// TIA Portal project "Proyecto_Dosificador_Mezclador_Automatico" (V17)

(* hardware
DEVICE "S7-1200 station_1"  S7-1200 Station
   slot 0: "Rack_0"  S7-1200 Rack  Rack  V1.0
   slot 1: "PLC_1"  CPU 1215C DC/DC/DC  6ES7 215-1AG40-0XB0  V4.5
*)

// ===== PLC "PLC_1"  CPU 1215C DC/DC/DC =====

VAR_GLOBAL   // PLC tag table "Default tag table"
   "System_Byte" AT %MB8190 : Byte;
   "FirstScan" AT %M8190.0 : Bool;
   "DiagStatusUpdate" AT %M8190.1 : Bool;
   "AlwaysTRUE" AT %M8190.2 : Bool;
   "AlwaysFALSE" AT %M8190.3 : Bool;
   "Clock_Byte" AT %MB8191 : Byte;
   "Clock_10Hz" AT %M8191.0 : Bool;
   "Clock_5Hz" AT %M8191.1 : Bool;
   "Clock_2.5Hz" AT %M8191.2 : Bool;
   "Clock_2Hz" AT %M8191.3 : Bool;
   "Clock_1.25Hz" AT %M8191.4 : Bool;
   "Clock_1Hz" AT %M8191.5 : Bool;
   "Clock_0.625Hz" AT %M8191.6 : Bool;
   "Clock_0.5Hz" AT %M8191.7 : Bool;
END_VAR

VAR_GLOBAL   // PLC tag table "Entradas"
   "Sel Funcionamiento" AT %I0.0 : Bool;
   "P Marcha NO" AT %I0.1 : Bool;
   "P Paro NC" AT %I0.2 : Bool;
   "P Emergencia NC" AT %I0.3 : Bool;
   "P Rearme NO" AT %I0.4 : Bool;
   "S Mezclador Nivel Bajo NC" AT %I0.5 : Bool;
   "S Briquetas NO" AT %I0.6 : Bool;
   "S FC Pivotante Arriba NC" AT %I0.7 : Bool;
   "S FC Pivotante Abajo NC" AT %I1.0 : Bool;
   "GM Cinta NC" AT %I1.1 : Bool;
   "GM Agitador NC" AT %I1.2 : Bool;
   "GM Pivotante NC" AT %I1.3 : Bool;
   "S Peso" AT %IW64 : Word;
END_VAR

VAR_GLOBAL   // PLC tag table "Salidas"
   "EV A Monoestable NC" AT %I1.6 : Bool;
   "EV B Monoestable NC" AT %I1.7 : Bool;
   "EV C Monoestable NC" AT %I2.0 : Bool;
   "M Cinta" AT %I2.1 : Bool;
   "M Agitador" AT %I2.2 : Bool;
   "M Pivotante Subir" AT %I2.3 : Bool;
   "M Pivotante Bajar" AT %I2.4 : Bool;
END_VAR

VAR_GLOBAL   // PLC tag table "Marcas Generales"
   "S Peso Normalizado" AT %MD2000 : Real;
   "S Peso Escalado" AT %MD2004 : Real;
   "Marca Marcha NO" AT %M2008.0 : Bool;
   "Marca Paro NC" AT %M2008.1 : Bool;
   "Marca Seguridad NC" AT %M2008.2 : Bool;
   "Marca Rearme NO" AT %M2008.3 : Bool;
   "Marca Sel Funcionamiento" AT %M2008.4 : Bool;
   "Marca Sel Mantenimiento" AT %M2008.5 : Bool;
   "Marca CI Todas" AT %M2008.6 : Bool;
   "Marca Etapas Iniciales" AT %M2008.7 : Bool;
   "Marca CI Mezclador" AT %M2009.0 : Bool;
   "Marca CI Depositos" AT %M2009.1 : Bool;
   "Marca CI Briquetas" AT %M2009.2 : Bool;
   "Marca CI Electrovalvulas" AT %M2009.3 : Bool;
END_VAR

VAR_GLOBAL   // PLC tag table "Etapas"
   "E0" AT %M0.0 : Bool;   // Etapas funcionamiento E0-E99
   "E1" AT %M0.1 : Bool;   // Etapas funcionamiento E0-E99
   "E2" AT %M0.2 : Bool;   // Etapas funcionamiento E0-E99
   "E3" AT %M0.3 : Bool;   // Etapas funcionamiento E0-E99
   "E4" AT %M0.4 : Bool;   // Etapas funcionamiento E0-E99
   "E5" AT %M0.5 : Bool;   // Etapas funcionamiento E0-E99
   "E6" AT %M0.6 : Bool;   // Etapas funcionamiento E0-E99
   "E7" AT %M0.7 : Bool;   // Etapas funcionamiento E0-E99
   "E8" AT %M1.0 : Bool;   // Etapas funcionamiento E0-E99
   "E9" AT %M1.1 : Bool;   // Etapas funcionamiento E0-E99
   "E10" AT %M1.2 : Bool;   // Etapas funcionamiento E0-E99
   "E11" AT %M1.3 : Bool;   // Etapas funcionamiento E0-E99
   "E12" AT %M1.4 : Bool;   // Etapas funcionamiento E0-E99
   "E13" AT %M1.5 : Bool;   // Etapas funcionamiento E0-E99
   "E14" AT %M1.6 : Bool;   // Etapas funcionamiento E0-E99
   "E15" AT %M1.7 : Bool;   // Etapas funcionamiento E0-E99
   "E16" AT %M2.0 : Bool;   // Etapas funcionamiento E0-E99
   "E17" AT %M2.1 : Bool;   // Etapas funcionamiento E0-E99
   "E18" AT %M2.2 : Bool;   // Etapas funcionamiento E0-E99
   "E19" AT %M2.3 : Bool;   // Etapas funcionamiento E0-E99
   "E20" AT %M2.4 : Bool;   // Etapas funcionamiento E0-E99
   "E21" AT %M2.5 : Bool;   // Etapas funcionamiento E0-E99
   "E22" AT %M2.6 : Bool;   // Etapas funcionamiento E0-E99
   "E23" AT %M2.7 : Bool;   // Etapas funcionamiento E0-E99
   "E24" AT %M3.0 : Bool;   // Etapas funcionamiento E0-E99
   "E25" AT %M3.1 : Bool;   // Etapas funcionamiento E0-E99
   "E26" AT %M3.2 : Bool;   // Etapas funcionamiento E0-E99
   "E27" AT %M3.3 : Bool;   // Etapas funcionamiento E0-E99
   "E28" AT %M3.4 : Bool;   // Etapas funcionamiento E0-E99
   "E29" AT %M3.5 : Bool;   // Etapas funcionamiento E0-E99
   "E30" AT %M3.6 : Bool;   // Etapas funcionamiento E0-E99
   "E31" AT %M3.7 : Bool;   // Etapas funcionamiento E0-E99
   "E32" AT %M4.0 : Bool;   // Etapas funcionamiento E0-E99
   "E33" AT %M4.1 : Bool;   // Etapas funcionamiento E0-E99
   "E34" AT %M4.2 : Bool;   // Etapas funcionamiento E0-E99
   "E35" AT %M4.3 : Bool;   // Etapas funcionamiento E0-E99
   "E36" AT %M4.4 : Bool;   // Etapas funcionamiento E0-E99
   "E37" AT %M4.5 : Bool;   // Etapas funcionamiento E0-E99
   "E38" AT %M4.6 : Bool;   // Etapas funcionamiento E0-E99
   "E39" AT %M4.7 : Bool;   // Etapas funcionamiento E0-E99
   "E40" AT %M5.0 : Bool;   // Etapas funcionamiento E0-E99
   "E41" AT %M5.1 : Bool;   // Etapas funcionamiento E0-E99
   "E42" AT %M5.2 : Bool;   // Etapas funcionamiento E0-E99
   "E43" AT %M5.3 : Bool;   // Etapas funcionamiento E0-E99
   "E44" AT %M5.4 : Bool;   // Etapas funcionamiento E0-E99
   "E45" AT %M5.5 : Bool;   // Etapas funcionamiento E0-E99
   "E46" AT %M5.6 : Bool;   // Etapas funcionamiento E0-E99
   "E47" AT %M5.7 : Bool;   // Etapas funcionamiento E0-E99
   "E48" AT %M6.0 : Bool;   // Etapas funcionamiento E0-E99
   "E49" AT %M6.1 : Bool;   // Etapas funcionamiento E0-E99
   "E50" AT %M6.2 : Bool;   // Etapas funcionamiento E0-E99
   "E51" AT %M6.3 : Bool;   // Etapas funcionamiento E0-E99
   "E52" AT %M6.4 : Bool;   // Etapas funcionamiento E0-E99
   "E53" AT %M6.5 : Bool;   // Etapas funcionamiento E0-E99
   "E54" AT %M6.6 : Bool;   // Etapas funcionamiento E0-E99
   "E55" AT %M6.7 : Bool;   // Etapas funcionamiento E0-E99
   "E56" AT %M7.0 : Bool;   // Etapas funcionamiento E0-E99
   "E57" AT %M7.1 : Bool;   // Etapas funcionamiento E0-E99
   "E58" AT %M7.2 : Bool;   // Etapas funcionamiento E0-E99
   "E59" AT %M7.3 : Bool;   // Etapas funcionamiento E0-E99
   "E60" AT %M7.4 : Bool;   // Etapas funcionamiento E0-E99
   "E61" AT %M7.5 : Bool;   // Etapas funcionamiento E0-E99
   "E62" AT %M7.6 : Bool;   // Etapas funcionamiento E0-E99
   "E63" AT %M7.7 : Bool;   // Etapas funcionamiento E0-E99
   "E64" AT %M8.0 : Bool;   // Etapas funcionamiento E0-E99
   "E65" AT %M8.1 : Bool;   // Etapas funcionamiento E0-E99
   "E66" AT %M8.2 : Bool;   // Etapas funcionamiento E0-E99
   "E67" AT %M8.3 : Bool;   // Etapas funcionamiento E0-E99
   "E68" AT %M8.4 : Bool;   // Etapas funcionamiento E0-E99
   "E69" AT %M8.5 : Bool;   // Etapas funcionamiento E0-E99
   "E70" AT %M8.6 : Bool;   // Etapas funcionamiento E0-E99
   "E71" AT %M8.7 : Bool;   // Etapas funcionamiento E0-E99
   "E72" AT %M9.0 : Bool;   // Etapas funcionamiento E0-E99
   "E73" AT %M9.1 : Bool;   // Etapas funcionamiento E0-E99
   "E74" AT %M9.2 : Bool;   // Etapas funcionamiento E0-E99
   "E75" AT %M9.3 : Bool;   // Etapas funcionamiento E0-E99
   "E76" AT %M9.4 : Bool;   // Etapas funcionamiento E0-E99
   "E77" AT %M9.5 : Bool;   // Etapas funcionamiento E0-E99
   "E78" AT %M9.6 : Bool;   // Etapas funcionamiento E0-E99
   "E79" AT %M9.7 : Bool;   // Etapas funcionamiento E0-E99
   "E80" AT %M10.0 : Bool;   // Etapas funcionamiento E0-E99
   "E81" AT %M10.1 : Bool;   // Etapas funcionamiento E0-E99
   "E82" AT %M10.2 : Bool;   // Etapas funcionamiento E0-E99
   "E83" AT %M10.3 : Bool;   // Etapas funcionamiento E0-E99
   "E84" AT %M10.4 : Bool;   // Etapas funcionamiento E0-E99
   "E85" AT %M10.5 : Bool;   // Etapas funcionamiento E0-E99
   "E86" AT %M10.6 : Bool;   // Etapas funcionamiento E0-E99
   "E87" AT %M10.7 : Bool;   // Etapas funcionamiento E0-E99
   "E88" AT %M11.0 : Bool;   // Etapas funcionamiento E0-E99
   "E89" AT %M11.1 : Bool;   // Etapas funcionamiento E0-E99
   "E90" AT %M11.2 : Bool;   // Etapas funcionamiento E0-E99
   "E91" AT %M11.3 : Bool;   // Etapas funcionamiento E0-E99
   "E92" AT %M11.4 : Bool;   // Etapas funcionamiento E0-E99
   "E93" AT %M11.5 : Bool;   // Etapas funcionamiento E0-E99
   "E94" AT %M11.6 : Bool;   // Etapas funcionamiento E0-E99
   "E95" AT %M11.7 : Bool;   // Etapas funcionamiento E0-E99
   "E96" AT %M12.0 : Bool;   // Etapas funcionamiento E0-E99
   "E97" AT %M12.1 : Bool;   // Etapas funcionamiento E0-E99
   "E98" AT %M12.2 : Bool;   // Etapas funcionamiento E0-E99
   "E99" AT %M12.3 : Bool;   // Etapas funcionamiento E0-E99
   "E100" AT %M100.0 : Bool;   // Etapas modos marcha E100-E199
   "E101" AT %M100.1 : Bool;   // Etapas modos marcha E100-E199
   "E102" AT %M100.2 : Bool;   // Etapas modos marcha E100-E199
   "E103" AT %M100.3 : Bool;   // Etapas modos marcha E100-E199
   "E104" AT %M100.4 : Bool;   // Etapas modos marcha E100-E199
   "E105" AT %M100.5 : Bool;   // Etapas modos marcha E100-E199
   "E106" AT %M100.6 : Bool;   // Etapas modos marcha E100-E199
   "E107" AT %M100.7 : Bool;   // Etapas modos marcha E100-E199
   "E108" AT %M101.0 : Bool;   // Etapas modos marcha E100-E199
   "E109" AT %M101.1 : Bool;   // Etapas modos marcha E100-E199
   "E110" AT %M101.2 : Bool;   // Etapas modos marcha E100-E199
   "E111" AT %M101.3 : Bool;   // Etapas modos marcha E100-E199
   "E112" AT %M101.4 : Bool;   // Etapas modos marcha E100-E199
   "E113" AT %M101.5 : Bool;   // Etapas modos marcha E100-E199
   "E114" AT %M101.6 : Bool;   // Etapas modos marcha E100-E199
   "E115" AT %M101.7 : Bool;   // Etapas modos marcha E100-E199
   "E116" AT %M102.0 : Bool;   // Etapas modos marcha E100-E199
   "E117" AT %M102.1 : Bool;   // Etapas modos marcha E100-E199
   "E118" AT %M102.2 : Bool;   // Etapas modos marcha E100-E199
   "E119" AT %M102.3 : Bool;   // Etapas modos marcha E100-E199
   "E120" AT %M102.4 : Bool;   // Etapas modos marcha E100-E199
   "E121" AT %M102.5 : Bool;   // Etapas modos marcha E100-E199
   "E122" AT %M102.6 : Bool;   // Etapas modos marcha E100-E199
   "E123" AT %M102.7 : Bool;   // Etapas modos marcha E100-E199
   "E124" AT %M103.0 : Bool;   // Etapas modos marcha E100-E199
   "E125" AT %M103.1 : Bool;   // Etapas modos marcha E100-E199
   "E126" AT %M103.2 : Bool;   // Etapas modos marcha E100-E199
   "E127" AT %M103.3 : Bool;   // Etapas modos marcha E100-E199
   "E128" AT %M103.4 : Bool;   // Etapas modos marcha E100-E199
   "E129" AT %M103.5 : Bool;   // Etapas modos marcha E100-E199
   "E130" AT %M103.6 : Bool;   // Etapas modos marcha E100-E199
   "E131" AT %M103.7 : Bool;   // Etapas modos marcha E100-E199
   "E132" AT %M104.0 : Bool;   // Etapas modos marcha E100-E199
   "E133" AT %M104.1 : Bool;   // Etapas modos marcha E100-E199
   "E134" AT %M104.2 : Bool;   // Etapas modos marcha E100-E199
   "E135" AT %M104.3 : Bool;   // Etapas modos marcha E100-E199
   "E136" AT %M104.4 : Bool;   // Etapas modos marcha E100-E199
   "E137" AT %M104.5 : Bool;   // Etapas modos marcha E100-E199
   "E138" AT %M104.6 : Bool;   // Etapas modos marcha E100-E199
   "E139" AT %M104.7 : Bool;   // Etapas modos marcha E100-E199
   "E140" AT %M105.0 : Bool;   // Etapas modos marcha E100-E199
   "E141" AT %M105.1 : Bool;   // Etapas modos marcha E100-E199
   "E142" AT %M105.2 : Bool;   // Etapas modos marcha E100-E199
   "E143" AT %M105.3 : Bool;   // Etapas modos marcha E100-E199
   "E144" AT %M105.4 : Bool;   // Etapas modos marcha E100-E199
   "E145" AT %M105.5 : Bool;   // Etapas modos marcha E100-E199
   "E146" AT %M105.6 : Bool;   // Etapas modos marcha E100-E199
   "E147" AT %M105.7 : Bool;   // Etapas modos marcha E100-E199
   "E148" AT %M106.0 : Bool;   // Etapas modos marcha E100-E199
   "E149" AT %M106.1 : Bool;   // Etapas modos marcha E100-E199
   "E150" AT %M106.2 : Bool;   // Etapas modos marcha E100-E199
   "E151" AT %M106.3 : Bool;   // Etapas modos marcha E100-E199
   "E152" AT %M106.4 : Bool;   // Etapas modos marcha E100-E199
   "E153" AT %M106.5 : Bool;   // Etapas modos marcha E100-E199
   "E154" AT %M106.6 : Bool;   // Etapas modos marcha E100-E199
   "E155" AT %M106.7 : Bool;   // Etapas modos marcha E100-E199
   "E156" AT %M107.0 : Bool;   // Etapas modos marcha E100-E199
   "E157" AT %M107.1 : Bool;   // Etapas modos marcha E100-E199
   "E158" AT %M107.2 : Bool;   // Etapas modos marcha E100-E199
   "E159" AT %M107.3 : Bool;   // Etapas modos marcha E100-E199
   "E160" AT %M107.4 : Bool;   // Etapas modos marcha E100-E199
   "E161" AT %M107.5 : Bool;   // Etapas modos marcha E100-E199
   "E162" AT %M107.6 : Bool;   // Etapas modos marcha E100-E199
   "E163" AT %M107.7 : Bool;   // Etapas modos marcha E100-E199
   "E164" AT %M108.0 : Bool;   // Etapas modos marcha E100-E199
   "E165" AT %M108.1 : Bool;   // Etapas modos marcha E100-E199
   "E166" AT %M108.2 : Bool;   // Etapas modos marcha E100-E199
   "E167" AT %M108.3 : Bool;   // Etapas modos marcha E100-E199
   "E168" AT %M108.4 : Bool;   // Etapas modos marcha E100-E199
   "E169" AT %M108.5 : Bool;   // Etapas modos marcha E100-E199
   "E170" AT %M108.6 : Bool;   // Etapas modos marcha E100-E199
   "E171" AT %M108.7 : Bool;   // Etapas modos marcha E100-E199
   "E172" AT %M109.0 : Bool;   // Etapas modos marcha E100-E199
   "E173" AT %M109.1 : Bool;   // Etapas modos marcha E100-E199
   "E174" AT %M109.2 : Bool;   // Etapas modos marcha E100-E199
   "E175" AT %M109.3 : Bool;   // Etapas modos marcha E100-E199
   "E176" AT %M109.4 : Bool;   // Etapas modos marcha E100-E199
   "E177" AT %M109.5 : Bool;   // Etapas modos marcha E100-E199
   "E178" AT %M109.6 : Bool;   // Etapas modos marcha E100-E199
   "E179" AT %M109.7 : Bool;   // Etapas modos marcha E100-E199
   "E180" AT %M110.0 : Bool;   // Etapas modos marcha E100-E199
   "E181" AT %M110.1 : Bool;   // Etapas modos marcha E100-E199
   "E182" AT %M110.2 : Bool;   // Etapas modos marcha E100-E199
   "E183" AT %M110.3 : Bool;   // Etapas modos marcha E100-E199
   "E184" AT %M110.4 : Bool;   // Etapas modos marcha E100-E199
   "E185" AT %M110.5 : Bool;   // Etapas modos marcha E100-E199
   "E186" AT %M110.6 : Bool;   // Etapas modos marcha E100-E199
   "E187" AT %M110.7 : Bool;   // Etapas modos marcha E100-E199
   "E188" AT %M111.0 : Bool;   // Etapas modos marcha E100-E199
   "E189" AT %M111.1 : Bool;   // Etapas modos marcha E100-E199
   "E190" AT %M111.2 : Bool;   // Etapas modos marcha E100-E199
   "E191" AT %M111.3 : Bool;   // Etapas modos marcha E100-E199
   "E192" AT %M111.4 : Bool;   // Etapas modos marcha E100-E199
   "E193" AT %M111.5 : Bool;   // Etapas modos marcha E100-E199
   "E194" AT %M111.6 : Bool;   // Etapas modos marcha E100-E199
   "E195" AT %M111.7 : Bool;   // Etapas modos marcha E100-E199
   "E196" AT %M112.0 : Bool;   // Etapas modos marcha E100-E199
   "E197" AT %M112.1 : Bool;   // Etapas modos marcha E100-E199
   "E198" AT %M112.2 : Bool;   // Etapas modos marcha E100-E199
   "E199" AT %M112.3 : Bool;   // Etapas modos marcha E100-E199
   "E200" AT %M200.0 : Bool;   // Etapas condiciones iniciales E200-E299
   "E201" AT %M200.1 : Bool;   // Etapas condiciones iniciales E200-E299
   "E202" AT %M200.2 : Bool;   // Etapas condiciones iniciales E200-E299
   "E203" AT %M200.3 : Bool;   // Etapas condiciones iniciales E200-E299
   "E204" AT %M200.4 : Bool;   // Etapas condiciones iniciales E200-E299
   "E205" AT %M200.5 : Bool;   // Etapas condiciones iniciales E200-E299
   "E206" AT %M200.6 : Bool;   // Etapas condiciones iniciales E200-E299
   "E207" AT %M200.7 : Bool;   // Etapas condiciones iniciales E200-E299
   "E208" AT %M201.0 : Bool;   // Etapas condiciones iniciales E200-E299
   "E209" AT %M201.1 : Bool;   // Etapas condiciones iniciales E200-E299
   "E210" AT %M201.2 : Bool;   // Etapas condiciones iniciales E200-E299
   "E211" AT %M201.3 : Bool;   // Etapas condiciones iniciales E200-E299
   "E212" AT %M201.4 : Bool;   // Etapas condiciones iniciales E200-E299
   "E213" AT %M201.5 : Bool;   // Etapas condiciones iniciales E200-E299
   "E214" AT %M201.6 : Bool;   // Etapas condiciones iniciales E200-E299
   "E215" AT %M201.7 : Bool;   // Etapas condiciones iniciales E200-E299
   "E216" AT %M202.0 : Bool;   // Etapas condiciones iniciales E200-E299
   "E217" AT %M202.1 : Bool;   // Etapas condiciones iniciales E200-E299
   "E218" AT %M202.2 : Bool;   // Etapas condiciones iniciales E200-E299
   "E219" AT %M202.3 : Bool;   // Etapas condiciones iniciales E200-E299
   "E220" AT %M202.4 : Bool;   // Etapas condiciones iniciales E200-E299
   "E221" AT %M202.5 : Bool;   // Etapas condiciones iniciales E200-E299
   "E222" AT %M202.6 : Bool;   // Etapas condiciones iniciales E200-E299
   "E223" AT %M202.7 : Bool;   // Etapas condiciones iniciales E200-E299
   "E224" AT %M203.0 : Bool;   // Etapas condiciones iniciales E200-E299
   "E225" AT %M203.1 : Bool;   // Etapas condiciones iniciales E200-E299
   "E226" AT %M203.2 : Bool;   // Etapas condiciones iniciales E200-E299
   "E227" AT %M203.3 : Bool;   // Etapas condiciones iniciales E200-E299
   "E228" AT %M203.4 : Bool;   // Etapas condiciones iniciales E200-E299
   "E229" AT %M203.5 : Bool;   // Etapas condiciones iniciales E200-E299
   "E230" AT %M203.6 : Bool;   // Etapas condiciones iniciales E200-E299
   "E231" AT %M203.7 : Bool;   // Etapas condiciones iniciales E200-E299
   "E232" AT %M204.0 : Bool;   // Etapas condiciones iniciales E200-E299
   "E233" AT %M204.1 : Bool;   // Etapas condiciones iniciales E200-E299
   "E234" AT %M204.2 : Bool;   // Etapas condiciones iniciales E200-E299
   "E235" AT %M204.3 : Bool;   // Etapas condiciones iniciales E200-E299
   "E236" AT %M204.4 : Bool;   // Etapas condiciones iniciales E200-E299
   "E237" AT %M204.5 : Bool;   // Etapas condiciones iniciales E200-E299
   "E238" AT %M204.6 : Bool;   // Etapas condiciones iniciales E200-E299
   "E239" AT %M204.7 : Bool;   // Etapas condiciones iniciales E200-E299
   "E240" AT %M205.0 : Bool;   // Etapas condiciones iniciales E200-E299
   "E241" AT %M205.1 : Bool;   // Etapas condiciones iniciales E200-E299
   "E242" AT %M205.2 : Bool;   // Etapas condiciones iniciales E200-E299
   "E243" AT %M205.3 : Bool;   // Etapas condiciones iniciales E200-E299
   "E244" AT %M205.4 : Bool;   // Etapas condiciones iniciales E200-E299
   "E245" AT %M205.5 : Bool;   // Etapas condiciones iniciales E200-E299
   "E246" AT %M205.6 : Bool;   // Etapas condiciones iniciales E200-E299
   "E247" AT %M205.7 : Bool;   // Etapas condiciones iniciales E200-E299
   "E248" AT %M206.0 : Bool;   // Etapas condiciones iniciales E200-E299
   "E249" AT %M206.1 : Bool;   // Etapas condiciones iniciales E200-E299
   "E250" AT %M206.2 : Bool;   // Etapas condiciones iniciales E200-E299
   "E251" AT %M206.3 : Bool;   // Etapas condiciones iniciales E200-E299
   "E252" AT %M206.4 : Bool;   // Etapas condiciones iniciales E200-E299
   "E253" AT %M206.5 : Bool;   // Etapas condiciones iniciales E200-E299
   "E254" AT %M206.6 : Bool;   // Etapas condiciones iniciales E200-E299
   "E255" AT %M206.7 : Bool;   // Etapas condiciones iniciales E200-E299
   "E256" AT %M207.0 : Bool;   // Etapas condiciones iniciales E200-E299
   "E257" AT %M207.1 : Bool;   // Etapas condiciones iniciales E200-E299
   "E258" AT %M207.2 : Bool;   // Etapas condiciones iniciales E200-E299
   "E259" AT %M207.3 : Bool;   // Etapas condiciones iniciales E200-E299
   "E260" AT %M207.4 : Bool;   // Etapas condiciones iniciales E200-E299
   "E261" AT %M207.5 : Bool;   // Etapas condiciones iniciales E200-E299
   "E262" AT %M207.6 : Bool;   // Etapas condiciones iniciales E200-E299
   "E263" AT %M207.7 : Bool;   // Etapas condiciones iniciales E200-E299
   "E264" AT %M208.0 : Bool;   // Etapas condiciones iniciales E200-E299
   "E265" AT %M208.1 : Bool;   // Etapas condiciones iniciales E200-E299
   "E266" AT %M208.2 : Bool;   // Etapas condiciones iniciales E200-E299
   "E267" AT %M208.3 : Bool;   // Etapas condiciones iniciales E200-E299
   "E268" AT %M208.4 : Bool;   // Etapas condiciones iniciales E200-E299
   "E269" AT %M208.5 : Bool;   // Etapas condiciones iniciales E200-E299
   "E270" AT %M208.6 : Bool;   // Etapas condiciones iniciales E200-E299
   "E271" AT %M208.7 : Bool;   // Etapas condiciones iniciales E200-E299
   "E272" AT %M209.0 : Bool;   // Etapas condiciones iniciales E200-E299
   "E273" AT %M209.1 : Bool;   // Etapas condiciones iniciales E200-E299
   "E274" AT %M209.2 : Bool;   // Etapas condiciones iniciales E200-E299
   "E275" AT %M209.3 : Bool;   // Etapas condiciones iniciales E200-E299
   "E276" AT %M209.4 : Bool;   // Etapas condiciones iniciales E200-E299
   "E277" AT %M209.5 : Bool;   // Etapas condiciones iniciales E200-E299
   "E278" AT %M209.6 : Bool;   // Etapas condiciones iniciales E200-E299
   "E279" AT %M209.7 : Bool;   // Etapas condiciones iniciales E200-E299
   "E280" AT %M210.0 : Bool;   // Etapas condiciones iniciales E200-E299
   "E281" AT %M210.1 : Bool;   // Etapas condiciones iniciales E200-E299
   "E282" AT %M210.2 : Bool;   // Etapas condiciones iniciales E200-E299
   "E283" AT %M210.3 : Bool;   // Etapas condiciones iniciales E200-E299
   "E284" AT %M210.4 : Bool;   // Etapas condiciones iniciales E200-E299
   "E285" AT %M210.5 : Bool;   // Etapas condiciones iniciales E200-E299
   "E286" AT %M210.6 : Bool;   // Etapas condiciones iniciales E200-E299
   "E287" AT %M210.7 : Bool;   // Etapas condiciones iniciales E200-E299
   "E288" AT %M211.0 : Bool;   // Etapas condiciones iniciales E200-E299
   "E289" AT %M211.1 : Bool;   // Etapas condiciones iniciales E200-E299
   "E290" AT %M211.2 : Bool;   // Etapas condiciones iniciales E200-E299
   "E291" AT %M211.3 : Bool;   // Etapas condiciones iniciales E200-E299
   "E292" AT %M211.4 : Bool;   // Etapas condiciones iniciales E200-E299
   "E293" AT %M211.5 : Bool;   // Etapas condiciones iniciales E200-E299
   "E294" AT %M211.6 : Bool;   // Etapas condiciones iniciales E200-E299
   "E295" AT %M211.7 : Bool;   // Etapas condiciones iniciales E200-E299
   "E296" AT %M212.0 : Bool;   // Etapas condiciones iniciales E200-E299
   "E297" AT %M212.1 : Bool;   // Etapas condiciones iniciales E200-E299
   "E298" AT %M212.2 : Bool;   // Etapas condiciones iniciales E200-E299
   "E299" AT %M212.3 : Bool;   // Etapas condiciones iniciales E200-E299
   "E300" AT %M300.0 : Bool;   // Etapas paro E300-E399
   "E301" AT %M300.1 : Bool;   // Etapas paro E300-E399
   "E302" AT %M300.2 : Bool;   // Etapas paro E300-E399
   "E303" AT %M300.3 : Bool;   // Etapas paro E300-E399
   "E304" AT %M300.4 : Bool;   // Etapas paro E300-E399
   "E305" AT %M300.5 : Bool;   // Etapas paro E300-E399
   "E306" AT %M300.6 : Bool;   // Etapas paro E300-E399
   "E307" AT %M300.7 : Bool;   // Etapas paro E300-E399
   "E308" AT %M301.0 : Bool;   // Etapas paro E300-E399
   "E309" AT %M301.1 : Bool;   // Etapas paro E300-E399
   "E310" AT %M301.2 : Bool;   // Etapas paro E300-E399
   "E311" AT %M301.3 : Bool;   // Etapas paro E300-E399
   "E312" AT %M301.4 : Bool;   // Etapas paro E300-E399
   "E313" AT %M301.5 : Bool;   // Etapas paro E300-E399
   "E314" AT %M301.6 : Bool;   // Etapas paro E300-E399
   "E315" AT %M301.7 : Bool;   // Etapas paro E300-E399
   "E316" AT %M302.0 : Bool;   // Etapas paro E300-E399
   "E317" AT %M302.1 : Bool;   // Etapas paro E300-E399
   "E318" AT %M302.2 : Bool;   // Etapas paro E300-E399
   "E319" AT %M302.3 : Bool;   // Etapas paro E300-E399
   "E320" AT %M302.4 : Bool;   // Etapas paro E300-E399
   "E321" AT %M302.5 : Bool;   // Etapas paro E300-E399
   "E322" AT %M302.6 : Bool;   // Etapas paro E300-E399
   "E323" AT %M302.7 : Bool;   // Etapas paro E300-E399
   "E324" AT %M303.0 : Bool;   // Etapas paro E300-E399
   "E325" AT %M303.1 : Bool;   // Etapas paro E300-E399
   "E326" AT %M303.2 : Bool;   // Etapas paro E300-E399
   "E327" AT %M303.3 : Bool;   // Etapas paro E300-E399
   "E328" AT %M303.4 : Bool;   // Etapas paro E300-E399
   "E329" AT %M303.5 : Bool;   // Etapas paro E300-E399
   "E330" AT %M303.6 : Bool;   // Etapas paro E300-E399
   "E331" AT %M303.7 : Bool;   // Etapas paro E300-E399
   "E332" AT %M304.0 : Bool;   // Etapas paro E300-E399
   "E333" AT %M304.1 : Bool;   // Etapas paro E300-E399
   "E334" AT %M304.2 : Bool;   // Etapas paro E300-E399
   "E335" AT %M304.3 : Bool;   // Etapas paro E300-E399
   "E336" AT %M304.4 : Bool;   // Etapas paro E300-E399
   "E337" AT %M304.5 : Bool;   // Etapas paro E300-E399
   "E338" AT %M304.6 : Bool;   // Etapas paro E300-E399
   "E339" AT %M304.7 : Bool;   // Etapas paro E300-E399
   "E340" AT %M305.0 : Bool;   // Etapas paro E300-E399
   "E341" AT %M305.1 : Bool;   // Etapas paro E300-E399
   "E342" AT %M305.2 : Bool;   // Etapas paro E300-E399
   "E343" AT %M305.3 : Bool;   // Etapas paro E300-E399
   "E344" AT %M305.4 : Bool;   // Etapas paro E300-E399
   "E345" AT %M305.5 : Bool;   // Etapas paro E300-E399
   "E346" AT %M305.6 : Bool;   // Etapas paro E300-E399
   "E347" AT %M305.7 : Bool;   // Etapas paro E300-E399
   "E348" AT %M306.0 : Bool;   // Etapas paro E300-E399
   "E349" AT %M306.1 : Bool;   // Etapas paro E300-E399
   "E350" AT %M306.2 : Bool;   // Etapas paro E300-E399
   "E351" AT %M306.3 : Bool;   // Etapas paro E300-E399
   "E352" AT %M306.4 : Bool;   // Etapas paro E300-E399
   "E353" AT %M306.5 : Bool;   // Etapas paro E300-E399
   "E354" AT %M306.6 : Bool;   // Etapas paro E300-E399
   "E355" AT %M306.7 : Bool;   // Etapas paro E300-E399
   "E356" AT %M307.0 : Bool;   // Etapas paro E300-E399
   "E357" AT %M307.1 : Bool;   // Etapas paro E300-E399
   "E358" AT %M307.2 : Bool;   // Etapas paro E300-E399
   "E359" AT %M307.3 : Bool;   // Etapas paro E300-E399
   "E360" AT %M307.4 : Bool;   // Etapas paro E300-E399
   "E361" AT %M307.5 : Bool;   // Etapas paro E300-E399
   "E362" AT %M307.6 : Bool;   // Etapas paro E300-E399
   "E363" AT %M307.7 : Bool;   // Etapas paro E300-E399
   "E364" AT %M308.0 : Bool;   // Etapas paro E300-E399
   "E365" AT %M308.1 : Bool;   // Etapas paro E300-E399
   "E366" AT %M308.2 : Bool;   // Etapas paro E300-E399
   "E367" AT %M308.3 : Bool;   // Etapas paro E300-E399
   "E368" AT %M308.4 : Bool;   // Etapas paro E300-E399
   "E369" AT %M308.5 : Bool;   // Etapas paro E300-E399
   "E370" AT %M308.6 : Bool;   // Etapas paro E300-E399
   "E371" AT %M308.7 : Bool;   // Etapas paro E300-E399
   "E372" AT %M309.0 : Bool;   // Etapas paro E300-E399
   "E373" AT %M309.1 : Bool;   // Etapas paro E300-E399
   "E374" AT %M309.2 : Bool;   // Etapas paro E300-E399
   "E375" AT %M309.3 : Bool;   // Etapas paro E300-E399
   "E376" AT %M309.4 : Bool;   // Etapas paro E300-E399
   "E377" AT %M309.5 : Bool;   // Etapas paro E300-E399
   "E378" AT %M309.6 : Bool;   // Etapas paro E300-E399
   "E379" AT %M309.7 : Bool;   // Etapas paro E300-E399
   "E380" AT %M310.0 : Bool;   // Etapas paro E300-E399
   "E381" AT %M310.1 : Bool;   // Etapas paro E300-E399
   "E382" AT %M310.2 : Bool;   // Etapas paro E300-E399
   "E383" AT %M310.3 : Bool;   // Etapas paro E300-E399
   "E384" AT %M310.4 : Bool;   // Etapas paro E300-E399
   "E385" AT %M310.5 : Bool;   // Etapas paro E300-E399
   "E386" AT %M310.6 : Bool;   // Etapas paro E300-E399
   "E387" AT %M310.7 : Bool;   // Etapas paro E300-E399
   "E388" AT %M311.0 : Bool;   // Etapas paro E300-E399
   "E389" AT %M311.1 : Bool;   // Etapas paro E300-E399
   "E390" AT %M311.2 : Bool;   // Etapas paro E300-E399
   "E391" AT %M311.3 : Bool;   // Etapas paro E300-E399
   "E392" AT %M311.4 : Bool;   // Etapas paro E300-E399
   "E393" AT %M311.5 : Bool;   // Etapas paro E300-E399
   "E394" AT %M311.6 : Bool;   // Etapas paro E300-E399
   "E395" AT %M311.7 : Bool;   // Etapas paro E300-E399
   "E396" AT %M312.0 : Bool;   // Etapas paro E300-E399
   "E397" AT %M312.1 : Bool;   // Etapas paro E300-E399
   "E398" AT %M312.2 : Bool;   // Etapas paro E300-E399
   "E399" AT %M312.3 : Bool;   // Etapas paro E300-E399
   "E400" AT %M400.0 : Bool;   // Etapas emergencia E400-E499
   "E401" AT %M400.1 : Bool;   // Etapas emergencia E400-E499
   "E402" AT %M400.2 : Bool;   // Etapas emergencia E400-E499
   "E403" AT %M400.3 : Bool;   // Etapas emergencia E400-E499
   "E404" AT %M400.4 : Bool;   // Etapas emergencia E400-E499
   "E405" AT %M400.5 : Bool;   // Etapas emergencia E400-E499
   "E406" AT %M400.6 : Bool;   // Etapas emergencia E400-E499
   "E407" AT %M400.7 : Bool;   // Etapas emergencia E400-E499
   "E408" AT %M401.0 : Bool;   // Etapas emergencia E400-E499
   "E409" AT %M401.1 : Bool;   // Etapas emergencia E400-E499
   "E410" AT %M401.2 : Bool;   // Etapas emergencia E400-E499
   "E411" AT %M401.3 : Bool;   // Etapas emergencia E400-E499
   "E412" AT %M401.4 : Bool;   // Etapas emergencia E400-E499
   "E413" AT %M401.5 : Bool;   // Etapas emergencia E400-E499
   "E414" AT %M401.6 : Bool;   // Etapas emergencia E400-E499
   "E415" AT %M401.7 : Bool;   // Etapas emergencia E400-E499
   "E416" AT %M402.0 : Bool;   // Etapas emergencia E400-E499
   "E417" AT %M402.1 : Bool;   // Etapas emergencia E400-E499
   "E418" AT %M402.2 : Bool;   // Etapas emergencia E400-E499
   "E419" AT %M402.3 : Bool;   // Etapas emergencia E400-E499
   "E420" AT %M402.4 : Bool;   // Etapas emergencia E400-E499
   "E421" AT %M402.5 : Bool;   // Etapas emergencia E400-E499
   "E422" AT %M402.6 : Bool;   // Etapas emergencia E400-E499
   "E423" AT %M402.7 : Bool;   // Etapas emergencia E400-E499
   "E424" AT %M403.0 : Bool;   // Etapas emergencia E400-E499
   "E425" AT %M403.1 : Bool;   // Etapas emergencia E400-E499
   "E426" AT %M403.2 : Bool;   // Etapas emergencia E400-E499
   "E427" AT %M403.3 : Bool;   // Etapas emergencia E400-E499
   "E428" AT %M403.4 : Bool;   // Etapas emergencia E400-E499
   "E429" AT %M403.5 : Bool;   // Etapas emergencia E400-E499
   "E430" AT %M403.6 : Bool;   // Etapas emergencia E400-E499
   "E431" AT %M403.7 : Bool;   // Etapas emergencia E400-E499
   "E432" AT %M404.0 : Bool;   // Etapas emergencia E400-E499
   "E433" AT %M404.1 : Bool;   // Etapas emergencia E400-E499
   "E434" AT %M404.2 : Bool;   // Etapas emergencia E400-E499
   "E435" AT %M404.3 : Bool;   // Etapas emergencia E400-E499
   "E436" AT %M404.4 : Bool;   // Etapas emergencia E400-E499
   "E437" AT %M404.5 : Bool;   // Etapas emergencia E400-E499
   "E438" AT %M404.6 : Bool;   // Etapas emergencia E400-E499
   "E439" AT %M404.7 : Bool;   // Etapas emergencia E400-E499
   "E440" AT %M405.0 : Bool;   // Etapas emergencia E400-E499
   "E441" AT %M405.1 : Bool;   // Etapas emergencia E400-E499
   "E442" AT %M405.2 : Bool;   // Etapas emergencia E400-E499
   "E443" AT %M405.3 : Bool;   // Etapas emergencia E400-E499
   "E444" AT %M405.4 : Bool;   // Etapas emergencia E400-E499
   "E445" AT %M405.5 : Bool;   // Etapas emergencia E400-E499
   "E446" AT %M405.6 : Bool;   // Etapas emergencia E400-E499
   "E447" AT %M405.7 : Bool;   // Etapas emergencia E400-E499
   "E448" AT %M406.0 : Bool;   // Etapas emergencia E400-E499
   "E449" AT %M406.1 : Bool;   // Etapas emergencia E400-E499
   "E450" AT %M406.2 : Bool;   // Etapas emergencia E400-E499
   "E451" AT %M406.3 : Bool;   // Etapas emergencia E400-E499
   "E452" AT %M406.4 : Bool;   // Etapas emergencia E400-E499
   "E453" AT %M406.5 : Bool;   // Etapas emergencia E400-E499
   "E454" AT %M406.6 : Bool;   // Etapas emergencia E400-E499
   "E455" AT %M406.7 : Bool;   // Etapas emergencia E400-E499
   "E456" AT %M407.0 : Bool;   // Etapas emergencia E400-E499
   "E457" AT %M407.1 : Bool;   // Etapas emergencia E400-E499
   "E458" AT %M407.2 : Bool;   // Etapas emergencia E400-E499
   "E459" AT %M407.3 : Bool;   // Etapas emergencia E400-E499
   "E460" AT %M407.4 : Bool;   // Etapas emergencia E400-E499
   "E461" AT %M407.5 : Bool;   // Etapas emergencia E400-E499
   "E462" AT %M407.6 : Bool;   // Etapas emergencia E400-E499
   "E463" AT %M407.7 : Bool;   // Etapas emergencia E400-E499
   "E464" AT %M408.0 : Bool;   // Etapas emergencia E400-E499
   "E465" AT %M408.1 : Bool;   // Etapas emergencia E400-E499
   "E466" AT %M408.2 : Bool;   // Etapas emergencia E400-E499
   "E467" AT %M408.3 : Bool;   // Etapas emergencia E400-E499
   "E468" AT %M408.4 : Bool;   // Etapas emergencia E400-E499
   "E469" AT %M408.5 : Bool;   // Etapas emergencia E400-E499
   "E470" AT %M408.6 : Bool;   // Etapas emergencia E400-E499
   "E471" AT %M408.7 : Bool;   // Etapas emergencia E400-E499
   "E472" AT %M409.0 : Bool;   // Etapas emergencia E400-E499
   "E473" AT %M409.1 : Bool;   // Etapas emergencia E400-E499
   "E474" AT %M409.2 : Bool;   // Etapas emergencia E400-E499
   "E475" AT %M409.3 : Bool;   // Etapas emergencia E400-E499
   "E476" AT %M409.4 : Bool;   // Etapas emergencia E400-E499
   "E477" AT %M409.5 : Bool;   // Etapas emergencia E400-E499
   "E478" AT %M409.6 : Bool;   // Etapas emergencia E400-E499
   "E479" AT %M409.7 : Bool;   // Etapas emergencia E400-E499
   "E480" AT %M410.0 : Bool;   // Etapas emergencia E400-E499
   "E481" AT %M410.1 : Bool;   // Etapas emergencia E400-E499
   "E482" AT %M410.2 : Bool;   // Etapas emergencia E400-E499
   "E483" AT %M410.3 : Bool;   // Etapas emergencia E400-E499
   "E484" AT %M410.4 : Bool;   // Etapas emergencia E400-E499
   "E485" AT %M410.5 : Bool;   // Etapas emergencia E400-E499
   "E486" AT %M410.6 : Bool;   // Etapas emergencia E400-E499
   "E487" AT %M410.7 : Bool;   // Etapas emergencia E400-E499
   "E488" AT %M411.0 : Bool;   // Etapas emergencia E400-E499
   "E489" AT %M411.1 : Bool;   // Etapas emergencia E400-E499
   "E490" AT %M411.2 : Bool;   // Etapas emergencia E400-E499
   "E491" AT %M411.3 : Bool;   // Etapas emergencia E400-E499
   "E492" AT %M411.4 : Bool;   // Etapas emergencia E400-E499
   "E493" AT %M411.5 : Bool;   // Etapas emergencia E400-E499
   "E494" AT %M411.6 : Bool;   // Etapas emergencia E400-E499
   "E495" AT %M411.7 : Bool;   // Etapas emergencia E400-E499
   "E496" AT %M412.0 : Bool;   // Etapas emergencia E400-E499
   "E497" AT %M412.1 : Bool;   // Etapas emergencia E400-E499
   "E498" AT %M412.2 : Bool;   // Etapas emergencia E400-E499
   "E499" AT %M412.3 : Bool;   // Etapas emergencia E400-E499
   "E500" AT %M500.0 : Bool;   // Etapas mantenimiento E500-E599
   "E501" AT %M500.1 : Bool;   // Etapas mantenimiento E500-E599
   "E502" AT %M500.2 : Bool;   // Etapas mantenimiento E500-E599
   "E503" AT %M500.3 : Bool;   // Etapas mantenimiento E500-E599
   "E504" AT %M500.4 : Bool;   // Etapas mantenimiento E500-E599
   "E505" AT %M500.5 : Bool;   // Etapas mantenimiento E500-E599
   "E506" AT %M500.6 : Bool;   // Etapas mantenimiento E500-E599
   "E507" AT %M500.7 : Bool;   // Etapas mantenimiento E500-E599
   "E508" AT %M501.0 : Bool;   // Etapas mantenimiento E500-E599
   "E509" AT %M501.1 : Bool;   // Etapas mantenimiento E500-E599
   "E510" AT %M501.2 : Bool;   // Etapas mantenimiento E500-E599
   "E511" AT %M501.3 : Bool;   // Etapas mantenimiento E500-E599
   "E512" AT %M501.4 : Bool;   // Etapas mantenimiento E500-E599
   "E513" AT %M501.5 : Bool;   // Etapas mantenimiento E500-E599
   "E514" AT %M501.6 : Bool;   // Etapas mantenimiento E500-E599
   "E515" AT %M501.7 : Bool;   // Etapas mantenimiento E500-E599
   "E516" AT %M502.0 : Bool;   // Etapas mantenimiento E500-E599
   "E517" AT %M502.1 : Bool;   // Etapas mantenimiento E500-E599
   "E518" AT %M502.2 : Bool;   // Etapas mantenimiento E500-E599
   "E519" AT %M502.3 : Bool;   // Etapas mantenimiento E500-E599
   "E520" AT %M502.4 : Bool;   // Etapas mantenimiento E500-E599
   "E521" AT %M502.5 : Bool;   // Etapas mantenimiento E500-E599
   "E522" AT %M502.6 : Bool;   // Etapas mantenimiento E500-E599
   "E523" AT %M502.7 : Bool;   // Etapas mantenimiento E500-E599
   "E524" AT %M503.0 : Bool;   // Etapas mantenimiento E500-E599
   "E525" AT %M503.1 : Bool;   // Etapas mantenimiento E500-E599
   "E526" AT %M503.2 : Bool;   // Etapas mantenimiento E500-E599
   "E527" AT %M503.3 : Bool;   // Etapas mantenimiento E500-E599
   "E528" AT %M503.4 : Bool;   // Etapas mantenimiento E500-E599
   "E529" AT %M503.5 : Bool;   // Etapas mantenimiento E500-E599
   "E530" AT %M503.6 : Bool;   // Etapas mantenimiento E500-E599
   "E531" AT %M503.7 : Bool;   // Etapas mantenimiento E500-E599
   "E532" AT %M504.0 : Bool;   // Etapas mantenimiento E500-E599
   "E533" AT %M504.1 : Bool;   // Etapas mantenimiento E500-E599
   "E534" AT %M504.2 : Bool;   // Etapas mantenimiento E500-E599
   "E535" AT %M504.3 : Bool;   // Etapas mantenimiento E500-E599
   "E536" AT %M504.4 : Bool;   // Etapas mantenimiento E500-E599
   "E537" AT %M504.5 : Bool;   // Etapas mantenimiento E500-E599
   "E538" AT %M504.6 : Bool;   // Etapas mantenimiento E500-E599
   "E539" AT %M504.7 : Bool;   // Etapas mantenimiento E500-E599
   "E540" AT %M505.0 : Bool;   // Etapas mantenimiento E500-E599
   "E541" AT %M505.1 : Bool;   // Etapas mantenimiento E500-E599
   "E542" AT %M505.2 : Bool;   // Etapas mantenimiento E500-E599
   "E543" AT %M505.3 : Bool;   // Etapas mantenimiento E500-E599
   "E544" AT %M505.4 : Bool;   // Etapas mantenimiento E500-E599
   "E545" AT %M505.5 : Bool;   // Etapas mantenimiento E500-E599
   "E546" AT %M505.6 : Bool;   // Etapas mantenimiento E500-E599
   "E547" AT %M505.7 : Bool;   // Etapas mantenimiento E500-E599
   "E548" AT %M506.0 : Bool;   // Etapas mantenimiento E500-E599
   "E549" AT %M506.1 : Bool;   // Etapas mantenimiento E500-E599
   "E550" AT %M506.2 : Bool;   // Etapas mantenimiento E500-E599
   "E551" AT %M506.3 : Bool;   // Etapas mantenimiento E500-E599
   "E552" AT %M506.4 : Bool;   // Etapas mantenimiento E500-E599
   "E553" AT %M506.5 : Bool;   // Etapas mantenimiento E500-E599
   "E554" AT %M506.6 : Bool;   // Etapas mantenimiento E500-E599
   "E555" AT %M506.7 : Bool;   // Etapas mantenimiento E500-E599
   "E556" AT %M507.0 : Bool;   // Etapas mantenimiento E500-E599
   "E557" AT %M507.1 : Bool;   // Etapas mantenimiento E500-E599
   "E558" AT %M507.2 : Bool;   // Etapas mantenimiento E500-E599
   "E559" AT %M507.3 : Bool;   // Etapas mantenimiento E500-E599
   "E560" AT %M507.4 : Bool;   // Etapas mantenimiento E500-E599
   "E561" AT %M507.5 : Bool;   // Etapas mantenimiento E500-E599
   "E562" AT %M507.6 : Bool;   // Etapas mantenimiento E500-E599
   "E563" AT %M507.7 : Bool;   // Etapas mantenimiento E500-E599
   "E564" AT %M508.0 : Bool;   // Etapas mantenimiento E500-E599
   "E565" AT %M508.1 : Bool;   // Etapas mantenimiento E500-E599
   "E566" AT %M508.2 : Bool;   // Etapas mantenimiento E500-E599
   "E567" AT %M508.3 : Bool;   // Etapas mantenimiento E500-E599
   "E568" AT %M508.4 : Bool;   // Etapas mantenimiento E500-E599
   "E569" AT %M508.5 : Bool;   // Etapas mantenimiento E500-E599
   "E570" AT %M508.6 : Bool;   // Etapas mantenimiento E500-E599
   "E571" AT %M508.7 : Bool;   // Etapas mantenimiento E500-E599
   "E572" AT %M509.0 : Bool;   // Etapas mantenimiento E500-E599
   "E573" AT %M509.1 : Bool;   // Etapas mantenimiento E500-E599
   "E574" AT %M509.2 : Bool;   // Etapas mantenimiento E500-E599
   "E575" AT %M509.3 : Bool;   // Etapas mantenimiento E500-E599
   "E576" AT %M509.4 : Bool;   // Etapas mantenimiento E500-E599
   "E577" AT %M509.5 : Bool;   // Etapas mantenimiento E500-E599
   "E578" AT %M509.6 : Bool;   // Etapas mantenimiento E500-E599
   "E579" AT %M509.7 : Bool;   // Etapas mantenimiento E500-E599
   "E580" AT %M510.0 : Bool;   // Etapas mantenimiento E500-E599
   "E581" AT %M510.1 : Bool;   // Etapas mantenimiento E500-E599
   "E582" AT %M510.2 : Bool;   // Etapas mantenimiento E500-E599
   "E583" AT %M510.3 : Bool;   // Etapas mantenimiento E500-E599
   "E584" AT %M510.4 : Bool;   // Etapas mantenimiento E500-E599
   "E585" AT %M510.5 : Bool;   // Etapas mantenimiento E500-E599
   "E586" AT %M510.6 : Bool;   // Etapas mantenimiento E500-E599
   "E587" AT %M510.7 : Bool;   // Etapas mantenimiento E500-E599
   "E588" AT %M511.0 : Bool;   // Etapas mantenimiento E500-E599
   "E589" AT %M511.1 : Bool;   // Etapas mantenimiento E500-E599
   "E590" AT %M511.2 : Bool;   // Etapas mantenimiento E500-E599
   "E591" AT %M511.3 : Bool;   // Etapas mantenimiento E500-E599
   "E592" AT %M511.4 : Bool;   // Etapas mantenimiento E500-E599
   "E593" AT %M511.5 : Bool;   // Etapas mantenimiento E500-E599
   "E594" AT %M511.6 : Bool;   // Etapas mantenimiento E500-E599
   "E595" AT %M511.7 : Bool;   // Etapas mantenimiento E500-E599
   "E596" AT %M512.0 : Bool;   // Etapas mantenimiento E500-E599
   "E597" AT %M512.1 : Bool;   // Etapas mantenimiento E500-E599
   "E598" AT %M512.2 : Bool;   // Etapas mantenimiento E500-E599
   "E599" AT %M512.3 : Bool;   // Etapas mantenimiento E500-E599
END_VAR

VAR_GLOBAL   // PLC tag table "Variables proceso"
   "Posición peso 1" AT %MD800 : Real;
   "Posición peso 2" AT %MD804 : Real;
   "Posición peso 0" AT %MD808 : Real;
   "Flanco Briquetas" AT %M1000.0 : Bool;
END_VAR

// folder: System blocks/Program resources

DATA_BLOCK "T.ON 0"   // DB1
{ S7_Optimized_Access := 'TRUE' }
AUTHOR : Simatic
FAMILY : IEC
NAME : IEC_TMR
VERSION : 1.0
// stored: InstanceOfName IEC_TIMER
"IEC_TIMER"
BEGIN
END_DATA_BLOCK

DATA_BLOCK "Contador briquetas"   // DB2
{ S7_Optimized_Access := 'TRUE' }
AUTHOR : Simatic
FAMILY : IEC
NAME : CNTR
VERSION : 1.0
// stored: InstanceOfName IEC_COUNTER
"IEC_COUNTER"
BEGIN
END_DATA_BLOCK

// folder: (top level)

FUNCTION "EmergenciaEvolucion" : Void   // FC1, LAD
{ S7_Optimized_Access := 'TRUE' }
VERSION : 0.1
   VAR_TEMP   // added for the SCL form of the ladder/FBD networks
      _w1 : Bool;
   END_VAR
BEGIN

REGION Network 1: Etapas emergencia E400-E499
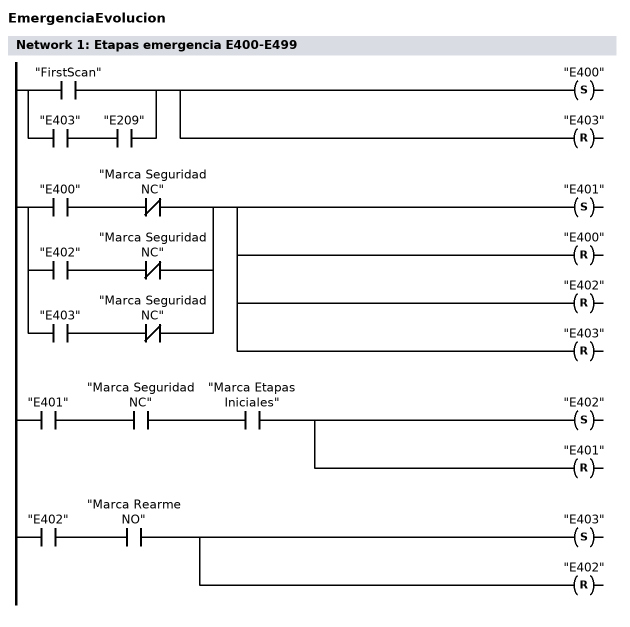
   RUNG wire#powerrail
      Contact( "FirstScan" )
      wire#w1
      S_Coil( "E400" )
   END_RUNG
   RUNG wire#powerrail
      Contact( "E403" )
      Contact( "E209" )
   END_RUNG wire#w1
   RUNG wire#w1
      R_Coil( "E403" )
   END_RUNG
   RUNG wire#powerrail
      Contact( "E400" )
      I_Contact( "Marca Seguridad NC" )
      wire#w2
      S_Coil( "E401" )
   END_RUNG
   RUNG wire#powerrail
      Contact( "E402" )
      I_Contact( "Marca Seguridad NC" )
   END_RUNG wire#w2
   RUNG wire#powerrail
      Contact( "E403" )
      I_Contact( "Marca Seguridad NC" )
   END_RUNG wire#w2
   RUNG wire#w2
      R_Coil( "E400" )
   END_RUNG
   RUNG wire#w2
      R_Coil( "E402" )
   END_RUNG
   RUNG wire#w2
      R_Coil( "E403" )
   END_RUNG
   RUNG wire#powerrail
      Contact( "E401" )
      Contact( "Marca Seguridad NC" )
      Contact( "Marca Etapas Iniciales" )
      wire#w3
      S_Coil( "E402" )
   END_RUNG
   RUNG wire#w3
      R_Coil( "E401" )
   END_RUNG
   RUNG wire#powerrail
      Contact( "E402" )
      Contact( "Marca Rearme NO" )
      wire#w4
      S_Coil( "E403" )
   END_RUNG
   RUNG wire#w4
      R_Coil( "E402" )
   END_RUNG
   // the same network as SCL:
   IF "FirstScan" OR ("E403" AND "E209") THEN
       "E400" := TRUE;
       "E403" := FALSE;
   END_IF;
   IF ("E400" AND NOT "Marca Seguridad NC") OR ("E402" AND NOT "Marca Seguridad NC") OR ("E403" AND NOT "Marca Seguridad NC") THEN
       "E401" := TRUE;
   END_IF;
   #_w1 := ("E400" AND NOT "Marca Seguridad NC") OR ("E402" AND NOT "Marca Seguridad NC") OR ("E403" AND NOT "Marca Seguridad NC");
   IF #_w1 THEN
       "E400" := FALSE;
       "E402" := FALSE;
       "E403" := FALSE;
   END_IF;
   IF "E401" AND "Marca Seguridad NC" AND "Marca Etapas Iniciales" THEN
       "E402" := TRUE;
       "E401" := FALSE;
   END_IF;
   IF "E402" AND "Marca Rearme NO" THEN
       "E403" := TRUE;
       "E402" := FALSE;
   END_IF;
END_REGION
END_FUNCTION

FUNCTION "Condiciones Iniciales" : Void   // FC2, LAD
{ S7_Optimized_Access := 'TRUE' }
VERSION : 0.1
BEGIN

REGION Network 1
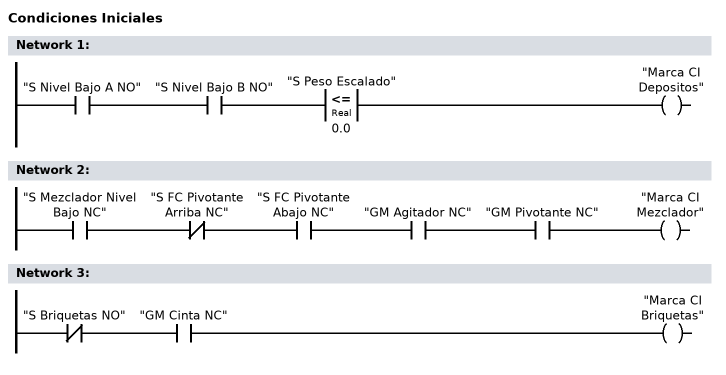
   RUNG wire#powerrail
      Contact( "S Nivel Bajo A NO" )
      Contact( "S Nivel Bajo B NO" )
      { S7_Templates := "SrcType := Real" } LE_Contact(in1 := "S Peso Escalado", in2 := 0.0)
      Coil( "Marca CI Depositos" )
   END_RUNG
   // the same network as SCL:
   "Marca CI Depositos" := "S Nivel Bajo A NO" AND "S Nivel Bajo B NO" AND ("S Peso Escalado" <= 0.0);
END_REGION

REGION Network 2
   RUNG wire#powerrail
      Contact( "S Mezclador Nivel Bajo NC" )
      I_Contact( "S FC Pivotante Arriba NC" )
      Contact( "S FC Pivotante Abajo NC" )
      Contact( "GM Agitador NC" )
      Contact( "GM Pivotante NC" )
      Coil( "Marca CI Mezclador" )
   END_RUNG
   // the same network as SCL:
   "Marca CI Mezclador" := "S Mezclador Nivel Bajo NC" AND NOT "S FC Pivotante Arriba NC" AND "S FC Pivotante Abajo NC" AND "GM Agitador NC" AND "GM Pivotante NC";
END_REGION

REGION Network 3
   RUNG wire#powerrail
      I_Contact( "S Briquetas NO" )
      Contact( "GM Cinta NC" )
      Coil( "Marca CI Briquetas" )
   END_RUNG
   // the same network as SCL:
   "Marca CI Briquetas" := NOT "S Briquetas NO" AND "GM Cinta NC";
END_REGION
END_FUNCTION

FUNCTION "Etapas Iniciales" : Void   // FC3, LAD
{ S7_Optimized_Access := 'TRUE' }
VERSION : 0.1
BEGIN
END_FUNCTION

FUNCTION "C. Iniciales Evolución" : Void   // FC4, LAD
{ S7_Optimized_Access := 'TRUE' }
VERSION : 0.1
   VAR_TEMP   // added for the SCL form of the ladder/FBD networks
      _w1 : Bool;
   END_VAR
BEGIN

REGION Network 1: Etapas condiciones iniciales E200-E299
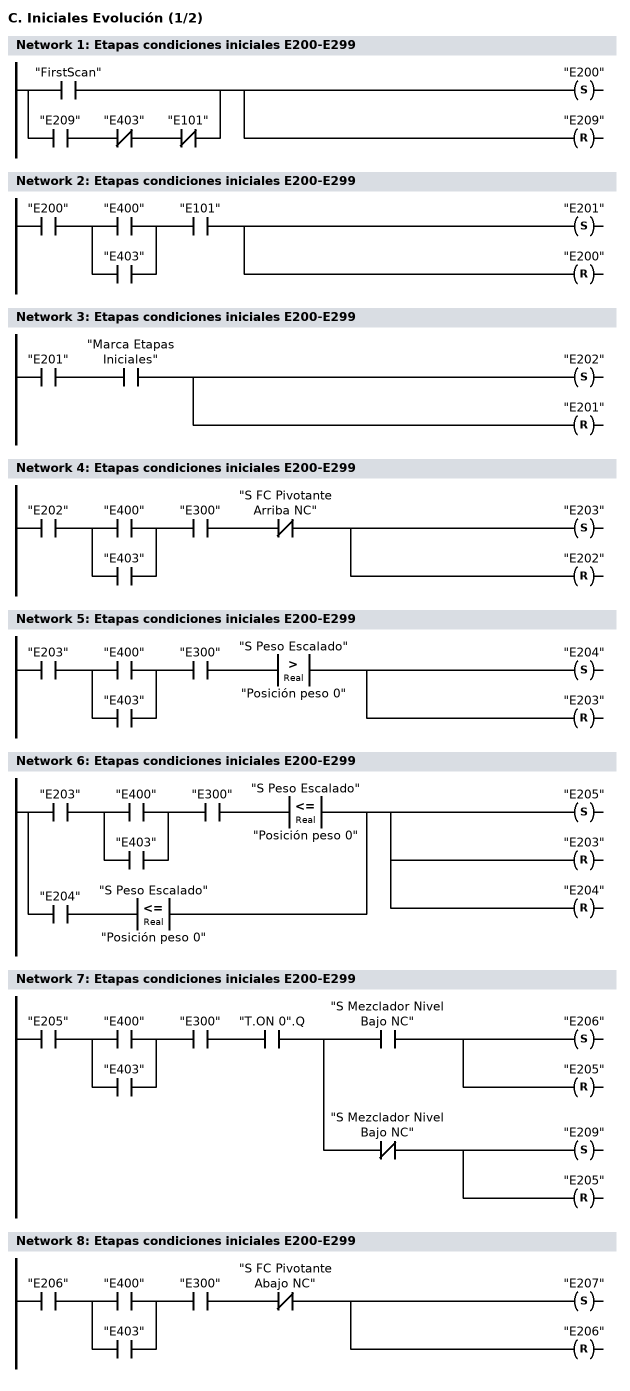
   RUNG wire#powerrail
      Contact( "FirstScan" )
      wire#w1
      S_Coil( "E200" )
   END_RUNG
   RUNG wire#powerrail
      Contact( "E209" )
      I_Contact( "E403" )
      I_Contact( "E101" )
   END_RUNG wire#w1
   RUNG wire#w1
      R_Coil( "E209" )
   END_RUNG
   // the same network as SCL:
   IF "FirstScan" OR ("E209" AND NOT "E403" AND NOT "E101") THEN
       "E200" := TRUE;
       "E209" := FALSE;
   END_IF;
END_REGION

REGION Network 2: Etapas condiciones iniciales E200-E299
   RUNG wire#powerrail
      Contact( "E200" )
      wire#w1
      Contact( "E400" )
      wire#w2
      Contact( "E101" )
      wire#w3
      S_Coil( "E201" )
   END_RUNG
   RUNG wire#w1
      Contact( "E403" )
   END_RUNG wire#w2
   RUNG wire#w3
      R_Coil( "E200" )
   END_RUNG
   // the same network as SCL:
   IF "E200" AND ("E400" OR "E403") AND "E101" THEN
       "E201" := TRUE;
       "E200" := FALSE;
   END_IF;
END_REGION

REGION Network 3: Etapas condiciones iniciales E200-E299
   RUNG wire#powerrail
      Contact( "E201" )
      Contact( "Marca Etapas Iniciales" )
      wire#w1
      S_Coil( "E202" )
   END_RUNG
   RUNG wire#w1
      R_Coil( "E201" )
   END_RUNG
   // the same network as SCL:
   IF "E201" AND "Marca Etapas Iniciales" THEN
       "E202" := TRUE;
       "E201" := FALSE;
   END_IF;
END_REGION

REGION Network 4: Etapas condiciones iniciales E200-E299
   RUNG wire#powerrail
      Contact( "E202" )
      wire#w1
      Contact( "E400" )
      wire#w2
      Contact( "E300" )
      I_Contact( "S FC Pivotante Arriba NC" )
      wire#w3
      S_Coil( "E203" )
   END_RUNG
   RUNG wire#w1
      Contact( "E403" )
   END_RUNG wire#w2
   RUNG wire#w3
      R_Coil( "E202" )
   END_RUNG
   // the same network as SCL:
   IF "E202" AND ("E400" OR "E403") AND "E300" AND NOT "S FC Pivotante Arriba NC" THEN
       "E203" := TRUE;
       "E202" := FALSE;
   END_IF;
END_REGION

REGION Network 5: Etapas condiciones iniciales E200-E299
   RUNG wire#powerrail
      Contact( "E203" )
      wire#w1
      Contact( "E400" )
      wire#w2
      Contact( "E300" )
      { S7_Templates := "SrcType := Real" } GT_Contact(in1 := "S Peso Escalado", in2 := "Posición peso 0")
      wire#w3
      S_Coil( "E204" )
   END_RUNG
   RUNG wire#w1
      Contact( "E403" )
   END_RUNG wire#w2
   RUNG wire#w3
      R_Coil( "E203" )
   END_RUNG
   // the same network as SCL:
   IF "E203" AND ("E400" OR "E403") AND "E300" AND ("S Peso Escalado" > "Posición peso 0") THEN
       "E204" := TRUE;
       "E203" := FALSE;
   END_IF;
END_REGION

REGION Network 6: Etapas condiciones iniciales E200-E299
   RUNG wire#powerrail
      Contact( "E203" )
      wire#w1
      Contact( "E400" )
      wire#w2
      Contact( "E300" )
      { S7_Templates := "SrcType := Real" } LE_Contact(in1 := "S Peso Escalado", in2 := "Posición peso 0")
      wire#w3
      S_Coil( "E205" )
   END_RUNG
   RUNG wire#w1
      Contact( "E403" )
   END_RUNG wire#w2
   RUNG wire#powerrail
      Contact( "E204" )
      { S7_Templates := "SrcType := Real" } LE_Contact(in1 := "S Peso Escalado", in2 := "Posición peso 0")
   END_RUNG wire#w3
   RUNG wire#w3
      R_Coil( "E203" )
   END_RUNG
   RUNG wire#w3
      R_Coil( "E204" )
   END_RUNG
   // the same network as SCL:
   IF ("E203" AND ("E400" OR "E403") AND "E300" AND ("S Peso Escalado" <= "Posición peso 0")) OR ("E204" AND ("S Peso Escalado" <= "Posición peso 0")) THEN
       "E205" := TRUE;
   END_IF;
   #_w1 := ("E203" AND ("E400" OR "E403") AND "E300" AND ("S Peso Escalado" <= "Posición peso 0")) OR ("E204" AND ("S Peso Escalado" <= "Posición peso 0"));
   IF #_w1 THEN
       "E203" := FALSE;
       "E204" := FALSE;
   END_IF;
END_REGION

REGION Network 7: Etapas condiciones iniciales E200-E299
   RUNG wire#powerrail
      Contact( "E205" )
      wire#w1
      Contact( "E400" )
      wire#w2
      Contact( "E300" )
      Contact( "T.ON 0".Q )
      wire#w3
      Contact( "S Mezclador Nivel Bajo NC" )
      wire#w4
      S_Coil( "E206" )
   END_RUNG
   RUNG wire#w1
      Contact( "E403" )
   END_RUNG wire#w2
   RUNG wire#w4
      R_Coil( "E205" )
   END_RUNG
   RUNG wire#w3
      I_Contact( "S Mezclador Nivel Bajo NC" )
      wire#w5
      S_Coil( "E209" )
   END_RUNG
   RUNG wire#w5
      R_Coil( "E205" )
   END_RUNG
   // the same network as SCL:
   #_w1 := "E205" AND ("E400" OR "E403") AND "E300" AND "T.ON 0".Q;
   IF #_w1 AND "S Mezclador Nivel Bajo NC" THEN
       "E206" := TRUE;
       "E205" := FALSE;
   END_IF;
   IF #_w1 AND NOT "S Mezclador Nivel Bajo NC" THEN
       "E209" := TRUE;
       "E205" := FALSE;
   END_IF;
END_REGION

REGION Network 8: Etapas condiciones iniciales E200-E299
   RUNG wire#powerrail
      Contact( "E206" )
      wire#w1
      Contact( "E400" )
      wire#w2
      Contact( "E300" )
      I_Contact( "S FC Pivotante Abajo NC" )
      wire#w3
      S_Coil( "E207" )
   END_RUNG
   RUNG wire#w1
      Contact( "E403" )
   END_RUNG wire#w2
   RUNG wire#w3
      R_Coil( "E206" )
   END_RUNG
   // the same network as SCL:
   IF "E206" AND ("E400" OR "E403") AND "E300" AND NOT "S FC Pivotante Abajo NC" THEN
       "E207" := TRUE;
       "E206" := FALSE;
   END_IF;
END_REGION

REGION Network 9: Etapas condiciones iniciales E200-E299
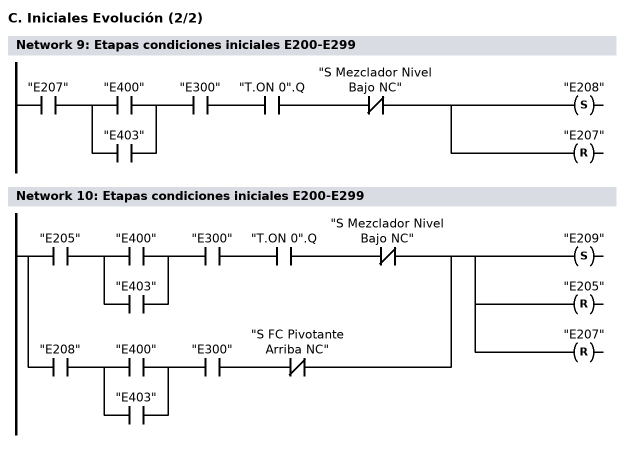
   RUNG wire#powerrail
      Contact( "E207" )
      wire#w1
      Contact( "E400" )
      wire#w2
      Contact( "E300" )
      Contact( "T.ON 0".Q )
      I_Contact( "S Mezclador Nivel Bajo NC" )
      wire#w3
      S_Coil( "E208" )
   END_RUNG
   RUNG wire#w1
      Contact( "E403" )
   END_RUNG wire#w2
   RUNG wire#w3
      R_Coil( "E207" )
   END_RUNG
   // the same network as SCL:
   IF "E207" AND ("E400" OR "E403") AND "E300" AND "T.ON 0".Q AND NOT "S Mezclador Nivel Bajo NC" THEN
       "E208" := TRUE;
       "E207" := FALSE;
   END_IF;
END_REGION

REGION Network 10: Etapas condiciones iniciales E200-E299
   RUNG wire#powerrail
      Contact( "E205" )
      wire#w1
      Contact( "E400" )
      wire#w2
      Contact( "E300" )
      Contact( "T.ON 0".Q )
      I_Contact( "S Mezclador Nivel Bajo NC" )
      wire#w3
      S_Coil( "E209" )
   END_RUNG
   RUNG wire#w1
      Contact( "E403" )
   END_RUNG wire#w2
   RUNG wire#powerrail
      Contact( "E208" )
      wire#w4
      Contact( "E400" )
      wire#w5
      Contact( "E300" )
      I_Contact( "S FC Pivotante Arriba NC" )
   END_RUNG wire#w3
   RUNG wire#w4
      Contact( "E403" )
   END_RUNG wire#w5
   RUNG wire#w3
      R_Coil( "E205" )
   END_RUNG
   RUNG wire#w3
      R_Coil( "E207" )
   END_RUNG
   // the same network as SCL:
   IF ("E205" AND ("E400" OR "E403") AND "E300" AND "T.ON 0".Q AND NOT "S Mezclador Nivel Bajo NC") OR ("E208" AND ("E400" OR "E403") AND "E300" AND NOT "S FC Pivotante Arriba NC") THEN
       "E209" := TRUE;
   END_IF;
   #_w1 := ("E205" AND ("E400" OR "E403") AND "E300" AND "T.ON 0".Q AND NOT "S Mezclador Nivel Bajo NC") OR ("E208" AND ("E400" OR "E403") AND "E300" AND NOT "S FC Pivotante Arriba NC");
   IF #_w1 THEN
       "E205" := FALSE;
       "E207" := FALSE;
   END_IF;
END_REGION
END_FUNCTION

FUNCTION "Funcionamiento Evolución" : Void   // FC5, LAD
{ S7_Optimized_Access := 'TRUE' }
VERSION : 0.1
   VAR_TEMP   // added for the SCL form of the ladder/FBD networks
      _w1 : Bool;
   END_VAR
BEGIN

REGION Network 1: Etapas funcionamiento E0-E99
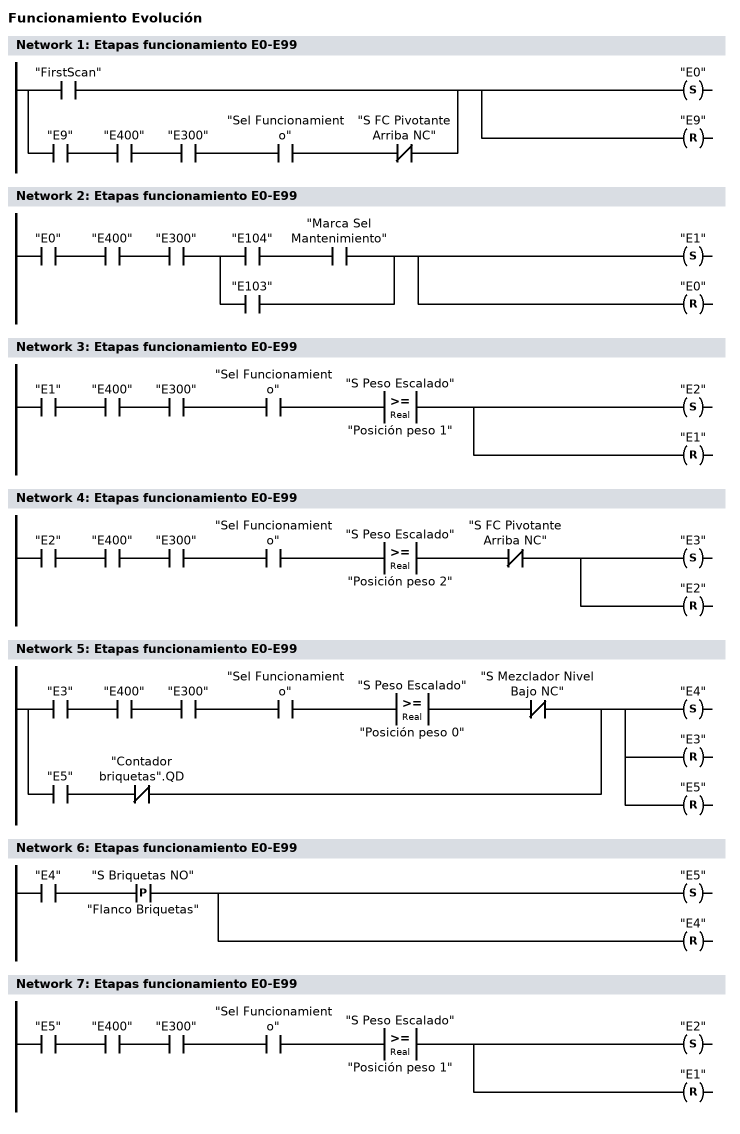
   RUNG wire#powerrail
      Contact( "FirstScan" )
      wire#w1
      S_Coil( "E0" )
   END_RUNG
   RUNG wire#powerrail
      Contact( "E9" )
      Contact( "E400" )
      Contact( "E300" )
      Contact( "Sel Funcionamiento" )
      I_Contact( "S FC Pivotante Arriba NC" )
   END_RUNG wire#w1
   RUNG wire#w1
      R_Coil( "E9" )
   END_RUNG
   // the same network as SCL:
   IF "FirstScan" OR ("E9" AND "E400" AND "E300" AND "Sel Funcionamiento" AND NOT "S FC Pivotante Arriba NC") THEN
       "E0" := TRUE;
       "E9" := FALSE;
   END_IF;
END_REGION

REGION Network 2: Etapas funcionamiento E0-E99
   RUNG wire#powerrail
      Contact( "E0" )
      Contact( "E400" )
      Contact( "E300" )
      wire#w1
      Contact( "E104" )
      Contact( "Marca Sel Mantenimiento" )
      wire#w2
      S_Coil( "E1" )
   END_RUNG
   RUNG wire#w1
      Contact( "E103" )
   END_RUNG wire#w2
   RUNG wire#w2
      R_Coil( "E0" )
   END_RUNG
   // the same network as SCL:
   IF "E0" AND "E400" AND "E300" AND (("E104" AND "Marca Sel Mantenimiento") OR "E103") THEN
       "E1" := TRUE;
       "E0" := FALSE;
   END_IF;
END_REGION

REGION Network 3: Etapas funcionamiento E0-E99
   RUNG wire#powerrail
      Contact( "E1" )
      Contact( "E400" )
      Contact( "E300" )
      Contact( "Sel Funcionamiento" )
      { S7_Templates := "SrcType := Real" } GE_Contact(in1 := "S Peso Escalado", in2 := "Posición peso 1")
      wire#w1
      S_Coil( "E2" )
   END_RUNG
   RUNG wire#w1
      R_Coil( "E1" )
   END_RUNG
   // the same network as SCL:
   IF "E1" AND "E400" AND "E300" AND "Sel Funcionamiento" AND ("S Peso Escalado" >= "Posición peso 1") THEN
       "E2" := TRUE;
       "E1" := FALSE;
   END_IF;
END_REGION

REGION Network 4: Etapas funcionamiento E0-E99
   RUNG wire#powerrail
      Contact( "E2" )
      Contact( "E400" )
      Contact( "E300" )
      Contact( "Sel Funcionamiento" )
      { S7_Templates := "SrcType := Real" } GE_Contact(in1 := "S Peso Escalado", in2 := "Posición peso 2")
      I_Contact( "S FC Pivotante Arriba NC" )
      wire#w1
      S_Coil( "E3" )
   END_RUNG
   RUNG wire#w1
      R_Coil( "E2" )
   END_RUNG
   // the same network as SCL:
   IF "E2" AND "E400" AND "E300" AND "Sel Funcionamiento" AND ("S Peso Escalado" >= "Posición peso 2") AND NOT "S FC Pivotante Arriba NC" THEN
       "E3" := TRUE;
       "E2" := FALSE;
   END_IF;
END_REGION

REGION Network 5: Etapas funcionamiento E0-E99
   RUNG wire#powerrail
      Contact( "E3" )
      Contact( "E400" )
      Contact( "E300" )
      Contact( "Sel Funcionamiento" )
      { S7_Templates := "SrcType := Real" } GE_Contact(in1 := "S Peso Escalado", in2 := "Posición peso 0")
      I_Contact( "S Mezclador Nivel Bajo NC" )
      wire#w1
      S_Coil( "E4" )
   END_RUNG
   RUNG wire#powerrail
      Contact( "E5" )
      I_Contact( "Contador briquetas".QD )
   END_RUNG wire#w1
   RUNG wire#w1
      R_Coil( "E3" )
   END_RUNG
   RUNG wire#w1
      R_Coil( "E5" )
   END_RUNG
   // the same network as SCL:
   IF ("E3" AND "E400" AND "E300" AND "Sel Funcionamiento" AND ("S Peso Escalado" >= "Posición peso 0") AND NOT "S Mezclador Nivel Bajo NC") OR ("E5" AND NOT "Contador briquetas".QD) THEN
       "E4" := TRUE;
   END_IF;
   #_w1 := ("E3" AND "E400" AND "E300" AND "Sel Funcionamiento" AND ("S Peso Escalado" >= "Posición peso 0") AND NOT "S Mezclador Nivel Bajo NC") OR ("E5" AND NOT "Contador briquetas".QD);
   IF #_w1 THEN
       "E3" := FALSE;
       "E5" := FALSE;
   END_IF;
END_REGION

REGION Network 6: Etapas funcionamiento E0-E99
   RUNG wire#powerrail
      Contact( "E4" )
      P_Contact(operand := "S Briquetas NO", bit := "Flanco Briquetas")
      wire#w1
      S_Coil( "E5" )
   END_RUNG
   RUNG wire#w1
      R_Coil( "E4" )
   END_RUNG
   // the same network as SCL:
   #_w1 := "E4" AND "S Briquetas NO" AND NOT "Flanco Briquetas";   // rising edge of "S Briquetas NO"
   "Flanco Briquetas" := "S Briquetas NO";
   IF #_w1 THEN
       "E5" := TRUE;
       "E4" := FALSE;
   END_IF;
END_REGION

REGION Network 7: Etapas funcionamiento E0-E99
   RUNG wire#powerrail
      Contact( "E5" )
      Contact( "E400" )
      Contact( "E300" )
      Contact( "Sel Funcionamiento" )
      { S7_Templates := "SrcType := Real" } GE_Contact(in1 := "S Peso Escalado", in2 := "Posición peso 1")
      wire#w1
      S_Coil( "E2" )
   END_RUNG
   RUNG wire#w1
      R_Coil( "E1" )
   END_RUNG
   // the same network as SCL:
   IF "E5" AND "E400" AND "E300" AND "Sel Funcionamiento" AND ("S Peso Escalado" >= "Posición peso 1") THEN
       "E2" := TRUE;
       "E1" := FALSE;
   END_IF;
END_REGION
END_FUNCTION

ORGANIZATION_BLOCK "Main"   // OB1, LAD, ProgramCycle
TITLE = "Main Program Sweep (Cycle)"
{ S7_Optimized_Access := 'TRUE' }
VERSION : 0.1
   VAR_INPUT
      Initial_Call : Bool;   // Initial call of this OB
      Remanence : Bool;   // =True, if remanent data are available
   END_VAR
BEGIN
END_ORGANIZATION_BLOCK